// TIA Portal V18 export
// export: Created 2025-12-01T17:50:35.5845931Z, ExportSetting None, DisplayName Totally Integrated Automation Portal, DisplayVersion V18 Update 5, DisplayName TIA Portal Openness, DisplayVersion V18 Update 5, DisplayName TIA Portal Teamcenter Gateway, DisplayVersion V18, DisplayName TIA Portal Version Control Interface, DisplayVersion V18, DisplayName STEP 7 Professional, DisplayVersion V18 Update 5, DisplayName STEP 7 Safety, DisplayVersion V18, DisplayName WinCC Professional, DisplayVersion V18 Update 5
DATA_BLOCK "ST10_PM"   // DB1063
{ S7_Optimized_Access := 'FALSE' }
// stored: AutoNumber false
   VAR RETAIN
      Num : Array[1..32] of "RCS_PMInterface_V1";
      Status { S7_SetPoint := 'True'} : Array[1..50] of Int;
   END_VAR
BEGIN
   // Num[1] : laszer marking
   // Num[2] : LabelFeeder
END_DATA_BLOCK
